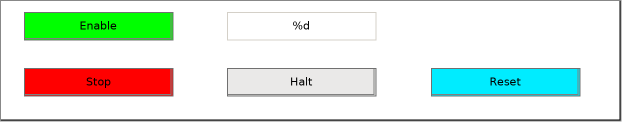
VISUALIZATION fAxis  // 622x122
VAR_IN_OUT
	io_fbAxis : Axis;
END_VAR
    Rectangle (0,0 620x120)
    Button (24,68 149x28), "Stop"
        tap io_fbAxis.bStop
    Textfield (227,12 149x28), "%d", text variable: io_fbAxis.axisRef.NcToPlc.AxisId
    Button (227,68 149x28), "Halt"
        tap io_fbAxis.bHalt
    Button (431,68 149x28), "Reset"
        tap io_fbAxis.bReset
    Button (24,12 149x28), "Enable"
        toggle io_fbAxis.bEnable
END_VISUALIZATION

(* stored: Version 1.1.0.1, ProductVersion 3.1.4024.2
   Visu fAxis: Id {9d9e460f-2c6c-4e8c-8893-340b4479a6c0} *)
